// TIA Portal project "SMART_FIFO_ARRAY" (V15)

(* hardware
DEVICE "S7-1200 station_1"  S7-1200 Station
   slot 0: "Rack_0"  S7-1200 Rack  Rack  V1.0
   slot 1: "PLC_1"  CPU 1217C DC/DC/DC  6ES7 217-1AG40-0XB0  V4.2
*)

// ===== PLC "PLC_1"  CPU 1217C DC/DC/DC =====

TYPE "FIFO_IO"
   STRUCT
      Din : DWord;
      "E" : Bool := true;
      RD : Bool;
      WD : Bool;
      RST : Bool;
      Dout : DWord;
      EMPTY : Bool := true;
      FULL : Bool;
      RD_Trigger : Bool;
      WD_Trigger : Bool;
   END_STRUCT;
END_TYPE

DATA_BLOCK "FIFO_Ver01_IDB_1"   // DB2
{ S7_Optimized_Access := 'TRUE' }
VERSION : 0.1
// stored: InstanceOfName FIFO_Ver01
"FIFO_Ver01"
BEGIN
END_DATA_BLOCK

DATA_BLOCK "GlobalDB_01"   // DB6
{ S7_Optimized_Access := 'TRUE' }
VERSION : 0.1
   VAR
      "FIFO_Ver01_IDB_IN/OUT" : "FIFO_IO";
      "FIFO_Ver01_IDB_IN/OUT_1" : "FIFO_IO";
   END_VAR
BEGIN
END_DATA_BLOCK

DATA_BLOCK "FIFO_Ver01_IDB_2"   // DB7
{ S7_Optimized_Access := 'TRUE' }
VERSION : 0.1
// stored: InstanceOfName FIFO_Ver01
"FIFO_Ver01"
BEGIN
END_DATA_BLOCK

FUNCTION_BLOCK "FIFO_Ver01"   // FB1, SCL
{ S7_Optimized_Access := 'TRUE' }
VERSION : 0.1
   VAR_INPUT
      Din : DWord;
      "E" : Bool := true;
      RD : Bool;
      POP : Int := 0;   // POP=1(standard POP); POP=2(POP+removal of similar elements from array)
      WD : Bool;
      RST : Bool;
   END_VAR
   VAR_OUTPUT
      Dout : DWord;
      EMPTY : Bool := true;
      FULL : Bool;
   END_VAR
   VAR
      fifo : Array[0..10] of DWord;
      pr_POP : Int;
      pr_no_POP : Int;
      pw : Int;
      pw_no_POP : Int;
      i : Int;
      j : Int;
      "counter" : Int;
   END_VAR
   VAR_TEMP
      k : Int;
   END_VAR
   VAR CONSTANT
      n : Int := 11;   // total number of elements in fifo array
   END_VAR
BEGIN
   //****************************EMPTY/FULL_POP
   IF #POP = 2 OR #POP=1 THEN
       #counter := 0;
       FOR #k := 0 TO #n DO
           IF #fifo[#k] <> 0 THEN
               #counter := #counter + 1;
           END_IF;
       END_FOR;
       IF #counter = #n THEN
           #FULL := TRUE;
       ELSE
           #FULL := FALSE;
       END_IF;

       IF #counter = 0 THEN
           #EMPTY := TRUE;
       ELSE
           #EMPTY := FALSE;
       END_IF;
   END_IF;


   //RESET
   IF #RST THEN
       #pw_no_POP := #pr_no_POP;
       #FULL := FALSE;
       #EMPTY := TRUE;
       #Dout := 0;
   //ENABLE    
   ELSIF #E THEN
       //****************************READ_POP=2
       IF NOT #EMPTY AND #POP=2 AND #RD THEN
           #Dout := #fifo[0];

           FOR #k := 0 TO #n DO
               IF #fifo[#k] = #Dout THEN
                   #fifo[#k] := 0;
               END_IF;
           END_FOR;

           FOR #i := 0 TO #n DO
               FOR #k := 0 TO #n - 1 DO
                   IF #fifo[#k] = 0 THEN
                       #fifo[#k] := #fifo[#k + 1];
                       #fifo[#k + 1] := 0;
                   END_IF;
               END_FOR;
           END_FOR;
       END_IF;


       //****************************READ_POP=1
       IF NOT #EMPTY AND #POP = 1 AND #RD THEN
           #Dout := #fifo[0];
           FOR #k := 0 TO #n - 1 DO
               #fifo[#k] := #fifo[#k + 1];
               #fifo[#k + 1] := 0;
           END_FOR;
       END_IF;


       //****************************READ_no POP 
       IF NOT #EMPTY AND #POP = 0 AND #RD THEN
           #Dout := #fifo[#pr_no_POP];
           IF #pr_no_POP >= #n - 1 THEN
               #pr_no_POP := 0;
           ELSE
               #pr_no_POP := #pr_no_POP + 1;
           END_IF;
           #EMPTY := #pr_no_POP = #pw_no_POP;
           #FULL := FALSE;
       END_IF;


       //****************************WRITE_POP    
       IF NOT #FULL AND (#POP=1 OR #POP=2) AND #WD THEN
           #counter := 0;
           FOR #k := 0 TO #n DO
               IF #fifo[#k] <> 0 THEN
                   #counter := #counter + 1;
               END_IF;
           END_FOR;

           #fifo[#counter] := #Din;
           #pw := #counter+1;
       END_IF;


       //****************************WRITE_no POP
       IF NOT #FULL AND #WD THEN
           #fifo[#pw_no_POP] := #Din;
           IF #pw_no_POP >= #n - 1 THEN
               #pw_no_POP := 0;
           ELSE
               #pw_no_POP := #pw_no_POP + 1;
           END_IF;
           #FULL := #pw_no_POP = #pr_no_POP;
           #EMPTY := FALSE;
       END_IF;

   END_IF;
END_FUNCTION_BLOCK

FUNCTION "INC1" : Void   // FC1, SCL
{ S7_Optimized_Access := 'TRUE' }
VERSION : 0.1
   VAR_INPUT
      X : Int;
      N : Int;
   END_VAR
   VAR_OUTPUT
      Out : Int;
   END_VAR
BEGIN
   IF #X >= #N - 1 THEN
       #Out := 0;
   ELSE
       #Out := #X + 1;
   END_IF;
END_FUNCTION

FUNCTION "POU(FC)_1" : Void   // FC100, FBD
{ S7_Optimized_Access := 'TRUE' }
VERSION : 0.1
BEGIN

REGION Network 1
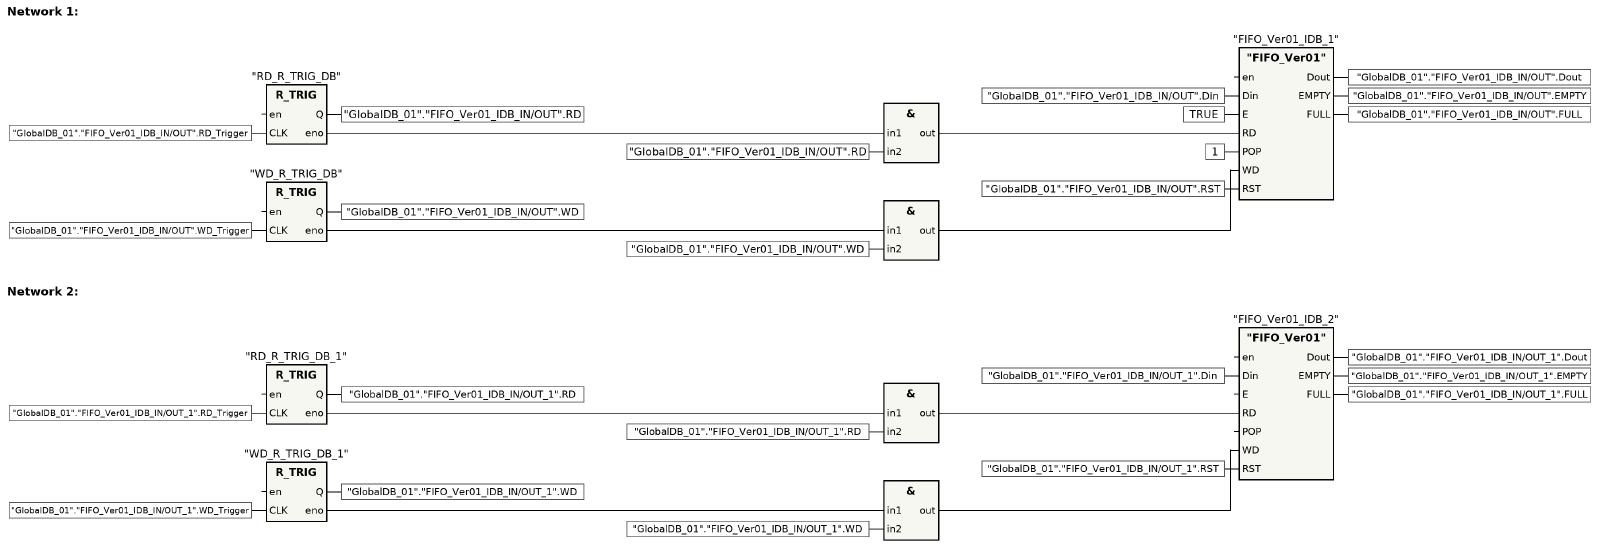
   // ENO of a box is taken as its EN; it also drops when the box reports an error
   "RD_R_TRIG_DB"(CLK := "GlobalDB_01"."FIFO_Ver01_IDB_IN/OUT".RD_Trigger,   // R_TRIG
                  Q => "GlobalDB_01"."FIFO_Ver01_IDB_IN/OUT".RD);
   "WD_R_TRIG_DB"(CLK := "GlobalDB_01"."FIFO_Ver01_IDB_IN/OUT".WD_Trigger,   // R_TRIG
                  Q => "GlobalDB_01"."FIFO_Ver01_IDB_IN/OUT".WD);
   "FIFO_Ver01_IDB_1"(Din := "GlobalDB_01"."FIFO_Ver01_IDB_IN/OUT".Din,   // "FIFO_Ver01"
                      "E" := TRUE,
                      RD := "GlobalDB_01"."FIFO_Ver01_IDB_IN/OUT".RD,
                      POP := 1,
                      WD := "GlobalDB_01"."FIFO_Ver01_IDB_IN/OUT".WD,
                      RST := "GlobalDB_01"."FIFO_Ver01_IDB_IN/OUT".RST,
                      Dout => "GlobalDB_01"."FIFO_Ver01_IDB_IN/OUT".Dout,
                      EMPTY => "GlobalDB_01"."FIFO_Ver01_IDB_IN/OUT".EMPTY,
                      FULL => "GlobalDB_01"."FIFO_Ver01_IDB_IN/OUT".FULL);
END_REGION

REGION Network 2
   // ENO of a box is taken as its EN; it also drops when the box reports an error
   "RD_R_TRIG_DB_1"(CLK := "GlobalDB_01"."FIFO_Ver01_IDB_IN/OUT_1".RD_Trigger,   // R_TRIG
                    Q => "GlobalDB_01"."FIFO_Ver01_IDB_IN/OUT_1".RD);
   "WD_R_TRIG_DB_1"(CLK := "GlobalDB_01"."FIFO_Ver01_IDB_IN/OUT_1".WD_Trigger,   // R_TRIG
                    Q => "GlobalDB_01"."FIFO_Ver01_IDB_IN/OUT_1".WD);
   "FIFO_Ver01_IDB_2"(Din := "GlobalDB_01"."FIFO_Ver01_IDB_IN/OUT_1".Din,   // "FIFO_Ver01"
                      RD := "GlobalDB_01"."FIFO_Ver01_IDB_IN/OUT_1".RD,
                      WD := "GlobalDB_01"."FIFO_Ver01_IDB_IN/OUT_1".WD,
                      RST := "GlobalDB_01"."FIFO_Ver01_IDB_IN/OUT_1".RST,
                      Dout => "GlobalDB_01"."FIFO_Ver01_IDB_IN/OUT_1".Dout,
                      EMPTY => "GlobalDB_01"."FIFO_Ver01_IDB_IN/OUT_1".EMPTY,
                      FULL => "GlobalDB_01"."FIFO_Ver01_IDB_IN/OUT_1".FULL);
END_REGION
END_FUNCTION

ORGANIZATION_BLOCK "Main"   // OB1, LAD, ProgramCycle
TITLE = "Main Program Sweep (Cycle)"
{ S7_Optimized_Access := 'TRUE' }
VERSION : 0.1
BEGIN

REGION Network 1
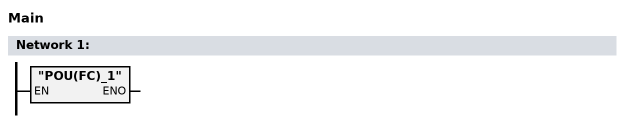
   RUNG wire#powerrail
      "POU(FC)_1"()
   END_RUNG
   // the same network as SCL:
   "POU(FC)_1"();
END_REGION
END_ORGANIZATION_BLOCK